FUNCTION_BLOCK LOAD_HMI (* XFER_HMI with Adapter *)
  (* Standard: 61499-1 *)
  (* Version 0.1, 2001-04-14, JHC, Rockwell Automation, Saved layout. *)
  (* Version 0.0, 2000-06-26, JHC, Rockwell Automation *)
  (* Compiler header: package fb.rt.omac; *)
  (* Compiler Java IBM VisualAge 3.0 *)
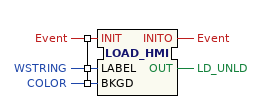
  EVENT_INPUT
    INIT WITH LABEL, BKGD; (* Initialization Request *)
  END_EVENT
  EVENT_OUTPUT
    INITO; (* Initialization Confirm *)
  END_EVENT
  VAR_INPUT
    LABEL : WSTRING := "LOAD";
    BKGD : COLOR := COLOR#blue; (* Background color when WO=0 *)
  END_VAR
  PLUGS
    OUT : LD_UNLD;
  END_PLUGS
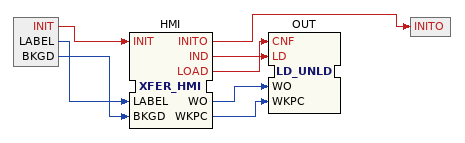
  FBS
    HMI : XFER_HMI;
  END_FBS
  EVENT_CONNECTIONS
    INIT TO HMI.INIT;
    HMI.INITO TO INITO;
    HMI.IND TO OUT.CNF;
    HMI.LOAD TO OUT.LD;
  END_CONNECTIONS
  DATA_CONNECTIONS
    LABEL TO HMI.LABEL;
    BKGD TO HMI.BKGD;
    HMI.WO TO OUT.WO;
    HMI.WKPC TO OUT.WKPC;
  END_CONNECTIONS
END_FUNCTION_BLOCK
